Yaskawa INFORM job: TCP_CHECK.JBI

/JOB
//NAME TCP_CHECK
//POS
///NPOS 4,0,0,1,0,0
///TOOL 0
///POSTYPE PULSE
///PULSE
C00000=-204317,-84436,-64683,-41499,-71625,29263
C00001=-204317,-90930,-87249,-44324,-63766,32764
C00002=-204317,-91143,-89097,-44673,-63021,33127
C00003=-204317,-84436,-64683,-41499,-71625,29263
///POSTYPE BASE
///RECTAN
///RCONF 1,0,0,0,0,0,0,0,0,0,0,0,0,0,0,0,0,0,0,0,0,0,0,0
P00100=275.000,0.000,875.000,180.0000,45.0000,0.0000
//INST
///DATE 2025/06/18 13:27
///ATTR SC,RW
///GROUP1 RB1
NOP
MOVJ P100 VJ=50.00
MOVJ C00000 VJ=30.00
MOVL C00001 V=211.7
MOVL C00002 V=10.6
PAUSE
MOVL C00003 V=211.7
MOVJ P100 VJ=50.00
END
